PROGRAM MAIN
VAR
    InheritanceRw : fbInheritanceLevel_5;
END_VAR

END_PROGRAM

(* stored: Version 1.1.0.1, ProductVersion 3.1.4024.6
   POU MAIN: Id {6d3b2b34-3b7b-4f9d-b63d-92fd87dfc156}, SpecialFunc None *)
